(* CODESYS project M241_LexiumILE_minimal_example.project
   Title: M241-ILS2K
   Version: 0.0.0.0
   Author: Philippe

Project tree, tasks and I/O mapping:
  MyController : TM241CE40R, Schneider Electric, order no. TM241CE40R, version 5.1.9.44
    application Application
      libraries: Integrated Lexium Library, 3.2.1.0 (Schneider Electric)
      task MAST (cyclic, interval 20 ms, priority 15, watchdog 100 ms x 1) calls ILE_functionblocks, DISABLE_LIMIT_SWITCH
      global variables GVL
      visualisation Visualization
      program ILE_functionblocks [FBD]
      program DISABLE_LIMIT_SWITCH [SFC]
    DI : Digital Inputs, Schneider Electric, version 5.1.9.44
        input  idwDI_IDW0 : DWORD  // IDW0
        input  ibDI_IB1 : BYTE  // IB1
    DQ : Digital Outputs, Schneider Electric, version 5.1.9.44
        output qwDQ_QW0 : WORD  // QW0
        output qbDQ_QB1 : BYTE  // QB1
    Counters : Counters, Schneider Electric, version 5.1.9.44
    Pulse_Generators : Pulse Generators, Schneider Electric, version 5.1.9.44
    Cartridge_1 : Cartridge, Schneider Electric, version 5.1.9.44
    Cartridge_2 : Cartridge, Schneider Electric, version 5.1.9.44
    IO_Bus : IO bus - TM3, Schneider Electric, version 5.1.9.44
    COM_Bus : COM bus, Schneider Electric, version 5.1.9.44
    Ethernet_1 : Ethernet Network, Schneider Electric, version 5.1.9.44
        settings: IPAddress = [192, 168, 100, 200]; SubnetMask = [255, 255, 255, 0]; GatewayAddress = [192, 168, 100, 254]; WebServer = TRUE; FTP Server = TRUE; SoMachine Protocol = TRUE; Modbus Server = TRUE; NetManage Protocol = TRUE; SNMP protocol = TRUE; Enable Routing = FALSE; WebVisu protocol = TRUE; DHCP Server Active = TRUE; Secured Web Server = TRUE
      Gestionnaire_Ethernet_Industriel : Industrial Ethernet Manager, Schneider Electric, version 1.0.12.40
          settings: BinaryFileSize = 586; Dhcps Host 0.Client Mac Address = [16#00, 16#80, 16#F4, 16#7B, 16#28, 16#E1]; Dhcps Host 0.Client Device Name = 'Lexium-ILx-002'; Dhcps Host 0.Client IP Address = [192, 168, 100, 159]; Dhcps Host 0.Network Mask = [255, 255, 255, 0]; Dhcps Host 0.Default Gateway = [192, 168, 100, 200]; Dhcps Host 2.Client Mac Address = [16#0, 16#0, 16#0, 16#0, 16#0]; Dhcps Host 3.Client Mac Address = [16#0, 16#0, 16#0, 16#0, 16#0]; Dhcps Host 4.Client Mac Address = [16#0, 16#0, 16#0, 16#0, 16#0]; Dhcps Host 5.Client Mac Address = [16#0, 16#0, 16#0, 16#0, 16#0]; Dhcps Host 6.Client Mac Address = [16#0, 16#0, 16#0, 16#0, 16#0]; Dhcps Host 7.Client Mac Address = [16#0, 16#0, 16#0, 16#0, 16#0]; Dhcps Host 8.Client Mac Address = [16#0, 16#0, 16#0, 16#0, 16#0]; Dhcps Host 9.Client Mac Address = [16#0, 16#0, 16#0, 16#0, 16#0]; Dhcps Host 10.Client Mac Address = [16#0, 16#0, 16#0, 16#0, 16#0]; Dhcps Host 11.Client Mac Address = [16#0, 16#0, 16#0, 16#0, 16#0]; Dhcps Host 12.Client Mac Address = [16#0, 16#0, 16#0, 16#0, 16#0]; Dhcps Host 13.Client Mac Address = [16#0, 16#0, 16#0, 16#0, 16#0]; Dhcps Host 14.Client Mac Address = [16#0, 16#0, 16#0, 16#0, 16#0]; Dhcps Host 15.Client Mac Address = [16#0, 16#0, 16#0, 16#0, 16#0]; Dhcps Host 16.Client Mac Address = [16#0, 16#0, 16#0, 16#0, 16#0]; Dhcps Host 17.Client Mac Address = [16#0, 16#0, 16#0, 16#0, 16#0]; Dhcps Host 18.Client Mac Address = [16#0, 16#0, 16#0, 16#0, 16#0]; Dhcps Host 19.Client Mac Address = [16#0, 16#0, 16#0, 16#0, 16#0]; Dhcps Host 20.Client Mac Address = [16#0, 16#0, 16#0, 16#0, 16#0]; Dhcps Host 21.Client Mac Address = [16#0, 16#0, 16#0, 16#0, 16#0]; Dhcps Host 22.Client Mac Address = [16#0, 16#0, 16#0, 16#0, 16#0]; Dhcps Host 23.Client Mac Address = [16#0, 16#0, 16#0, 16#0, 16#0]; Dhcps Host 24.Client Mac Address = [16#0, 16#0, 16#0, 16#0, 16#0]; Dhcps Host 25.Client Mac Address = [16#0, 16#0, 16#0, 16#0, 16#0]; Dhcps Host 26.Client Mac Address = [16#0, 16#0, 16#0, 16#0, 16#0]; Dhcps Host 27.Client Mac Address = [16#0, 16#0, 16#0, 16#0, 16#0]; Dhcps Host 28.Client Mac Address = [16#0, 16#0, 16#0, 16#0, 16#0]; Dhcps Host 29.Client Mac Address = [16#0, 16#0, 16#0, 16#0, 16#0]; Dhcps Host 30.Client Mac Address = [16#0, 16#0, 16#0, 16#0, 16#0]; Dhcps Host 31.Client Mac Address = [16#0, 16#0, 16#0, 16#0, 16#0]; Dhcps Host 32.Client Mac Address = [16#0, 16#0, 16#0, 16#0, 16#0]; Dhcps Host 33.Client Mac Address = [16#0, 16#0, 16#0, 16#0, 16#0]; Dhcps Host 34.Client Mac Address = [16#0, 16#0, 16#0, 16#0, 16#0]; Dhcps Host 35.Client Mac Address = [16#0, 16#0, 16#0, 16#0, 16#0];
            Dhcps Host 36.Client Mac Address = [16#0, 16#0, 16#0, 16#0, 16#0]; Dhcps Host 37.Client Mac Address = [16#0, 16#0, 16#0, 16#0, 16#0]; Dhcps Host 38.Client Mac Address = [16#0, 16#0, 16#0, 16#0, 16#0]; Dhcps Host 39.Client Mac Address = [16#0, 16#0, 16#0, 16#0, 16#0]; Dhcps Host 40.Client Mac Address = [16#0, 16#0, 16#0, 16#0, 16#0]; Dhcps Host 41.Client Mac Address = [16#0, 16#0, 16#0, 16#0, 16#0]; Dhcps Host 42.Client Mac Address = [16#0, 16#0, 16#0, 16#0, 16#0]; Dhcps Host 43.Client Mac Address = [16#0, 16#0, 16#0, 16#0, 16#0]; Dhcps Host 44.Client Mac Address = [16#0, 16#0, 16#0, 16#0, 16#0]; Dhcps Host 45.Client Mac Address = [16#0, 16#0, 16#0, 16#0, 16#0]; Dhcps Host 46.Client Mac Address = [16#0, 16#0, 16#0, 16#0, 16#0]; Dhcps Host 47.Client Mac Address = [16#0, 16#0, 16#0, 16#0, 16#0]; Dhcps Host 48.Client Mac Address = [16#0, 16#0, 16#0, 16#0, 16#0]; Dhcps Host 49.Client Mac Address = [16#0, 16#0, 16#0, 16#0, 16#0]; Dhcps Host 50.Client Mac Address = [16#0, 16#0, 16#0, 16#0, 16#0]; Dhcps Host 51.Client Mac Address = [16#0, 16#0, 16#0, 16#0, 16#0]; Dhcps Host 52.Client Mac Address = [16#0, 16#0, 16#0, 16#0, 16#0]; Dhcps Host 53.Client Mac Address = [16#0, 16#0, 16#0, 16#0, 16#0]; Dhcps Host 54.Client Mac Address = [16#0, 16#0, 16#0, 16#0, 16#0]; Dhcps Host 55.Client Mac Address = [16#0, 16#0, 16#0, 16#0, 16#0]; Dhcps Host 56.Client Mac Address = [16#0, 16#0, 16#0, 16#0, 16#0]; Dhcps Host 57.Client Mac Address = [16#0, 16#0, 16#0, 16#0, 16#0]; Dhcps Host 58.Client Mac Address = [16#0, 16#0, 16#0, 16#0, 16#0]; Dhcps Host 59.Client Mac Address = [16#0, 16#0, 16#0, 16#0, 16#0]; Dhcps Host 60.Client Mac Address = [16#0, 16#0, 16#0, 16#0, 16#0]; Dhcps Host 61.Client Mac Address = [16#0, 16#0, 16#0, 16#0, 16#0]; Dhcps Host 62.Client Mac Address = [16#0, 16#0, 16#0, 16#0, 16#0]; Dhcps Host 63.Client Mac Address = [16#0, 16#0, 16#0, 16#0, 16#0]; Dhcps Host 64.Client Mac Address = [16#0, 16#0, 16#0, 16#0, 16#0]; Dhcps Host 65.Client Mac Address = [16#0, 16#0, 16#0, 16#0, 16#0]; Dhcps Host 66.Client Mac Address = [16#0, 16#0, 16#0, 16#0, 16#0]; Dhcps Host 67.Client Mac Address = [16#0, 16#0, 16#0, 16#0, 16#0]; Dhcps Host 68.Client Mac Address = [16#0, 16#0, 16#0, 16#0, 16#0]; Dhcps Host 69.Client Mac Address = [16#0, 16#0, 16#0, 16#0, 16#0]; Dhcps Host 70.Client Mac Address = [16#0, 16#0, 16#0, 16#0, 16#0]; Dhcps Host 71.Client Mac Address = [16#0, 16#0, 16#0, 16#0, 16#0]; Dhcps Host 72.Client Mac Address = [16#0, 16#0, 16#0, 16#0, 16#0]; Dhcps Host 73.Client Mac Address = [16#0, 16#0, 16#0, 16#0, 16#0]; Dhcps Host 74.Client Mac Address = [16#0, 16#0, 16#0, 16#0, 16#0]; Dhcps Host 75.Client Mac Address = [16#0, 16#0, 16#0, 16#0, 16#0];
            Dhcps Host 76.Client Mac Address = [16#0, 16#0, 16#0, 16#0, 16#0]; Dhcps Host 77.Client Mac Address = [16#0, 16#0, 16#0, 16#0, 16#0]; Dhcps Host 78.Client Mac Address = [16#0, 16#0, 16#0, 16#0, 16#0]; Dhcps Host 79.Client Mac Address = [16#0, 16#0, 16#0, 16#0, 16#0]; Dhcps Host 80.Client Mac Address = [16#0, 16#0, 16#0, 16#0, 16#0]; Dhcps Host 81.Client Mac Address = [16#0, 16#0, 16#0, 16#0, 16#0]; Dhcps Host 82.Client Mac Address = [16#0, 16#0, 16#0, 16#0, 16#0]; Dhcps Host 83.Client Mac Address = [16#0, 16#0, 16#0, 16#0, 16#0]; Dhcps Host 84.Client Mac Address = [16#0, 16#0, 16#0, 16#0, 16#0]; Dhcps Host 85.Client Mac Address = [16#0, 16#0, 16#0, 16#0, 16#0]; Dhcps Host 86.Client Mac Address = [16#0, 16#0, 16#0, 16#0, 16#0]; Dhcps Host 87.Client Mac Address = [16#0, 16#0, 16#0, 16#0, 16#0]; Dhcps Host 88.Client Mac Address = [16#0, 16#0, 16#0, 16#0, 16#0]; Dhcps Host 89.Client Mac Address = [16#0, 16#0, 16#0, 16#0, 16#0]; Dhcps Host 90.Client Mac Address = [16#0, 16#0, 16#0, 16#0, 16#0]; Dhcps Host 91.Client Mac Address = [16#0, 16#0, 16#0, 16#0, 16#0]; Dhcps Host 92.Client Mac Address = [16#0, 16#0, 16#0, 16#0, 16#0]; Dhcps Host 93.Client Mac Address = [16#0, 16#0, 16#0, 16#0, 16#0]; Dhcps Host 94.Client Mac Address = [16#0, 16#0, 16#0, 16#0, 16#0]; Dhcps Host 95.Client Mac Address = [16#0, 16#0, 16#0, 16#0, 16#0]; Dhcps Host 96.Client Mac Address = [16#0, 16#0, 16#0, 16#0, 16#0]; Dhcps Host 97.Client Mac Address = [16#0, 16#0, 16#0, 16#0, 16#0]; Dhcps Host 98.Client Mac Address = [16#0, 16#0, 16#0, 16#0, 16#0]; Dhcps Host 99.Client Mac Address = [16#0, 16#0, 16#0, 16#0, 16#0]; Dhcps Host 100.Client Mac Address = [16#0, 16#0, 16#0, 16#0, 16#0]; Dhcps Host 101.Client Mac Address = [16#0, 16#0, 16#0, 16#0, 16#0]; Dhcps Host 102.Client Mac Address = [16#0, 16#0, 16#0, 16#0, 16#0]; Dhcps Host 103.Client Mac Address = [16#0, 16#0, 16#0, 16#0, 16#0]; Dhcps Host 104.Client Mac Address = [16#0, 16#0, 16#0, 16#0, 16#0]; Dhcps Host 105.Client Mac Address = [16#0, 16#0, 16#0, 16#0, 16#0]; Dhcps Host 106.Client Mac Address = [16#0, 16#0, 16#0, 16#0, 16#0]; Dhcps Host 107.Client Mac Address = [16#0, 16#0, 16#0, 16#0, 16#0]; Dhcps Host 108.Client Mac Address = [16#0, 16#0, 16#0, 16#0, 16#0]; Dhcps Host 109.Client Mac Address = [16#0, 16#0, 16#0, 16#0, 16#0]; Dhcps Host 110.Client Mac Address = [16#0, 16#0, 16#0, 16#0, 16#0]; Dhcps Host 111.Client Mac Address = [16#0, 16#0, 16#0, 16#0, 16#0]; Dhcps Host 112.Client Mac Address = [16#0, 16#0, 16#0, 16#0, 16#0]; Dhcps Host 113.Client Mac Address = [16#0, 16#0, 16#0, 16#0, 16#0]; Dhcps Host 114.Client Mac Address = [16#0, 16#0, 16#0, 16#0, 16#0]; Dhcps Host 115.Client Mac Address = [16#0, 16#0, 16#0, 16#0, 16#0];
            Dhcps Host 116.Client Mac Address = [16#0, 16#0, 16#0, 16#0, 16#0]; Dhcps Host 117.Client Mac Address = [16#0, 16#0, 16#0, 16#0, 16#0]; Dhcps Host 118.Client Mac Address = [16#0, 16#0, 16#0, 16#0, 16#0]; Dhcps Host 119.Client Mac Address = [16#0, 16#0, 16#0, 16#0, 16#0]; Dhcps Host 120.Client Mac Address = [16#0, 16#0, 16#0, 16#0, 16#0]; Dhcps Host 121.Client Mac Address = [16#0, 16#0, 16#0, 16#0, 16#0]; Dhcps Host 122.Client Mac Address = [16#0, 16#0, 16#0, 16#0, 16#0]; Dhcps Host 123.Client Mac Address = [16#0, 16#0, 16#0, 16#0, 16#0]; Dhcps Host 124.Client Mac Address = [16#0, 16#0, 16#0, 16#0, 16#0]; Dhcps Host 125.Client Mac Address = [16#0, 16#0, 16#0, 16#0, 16#0]; Dhcps Host 126.Client Mac Address = [16#0, 16#0, 16#0, 16#0, 16#0]; Dhcps Host 127.Client Mac Address = [16#0, 16#0, 16#0, 16#0, 16#0]; Dhcps Host 128.Client Mac Address = [16#0, 16#0, 16#0, 16#0, 16#0]; serialized Values = 010bc991-f7f9-45b2-8b15-1d199ae18604=0|; InterfaceUsedByDhcpSize = 4; InterfaceUsedByDhcp = [192,168,100,200]
          unmapped channels: Global Status, Healthbit 0, Healthbit 1, Healthbit 2, Healthbit 3, Channels 0, Channels 1, Channels 2, Channels 3
        Lexium_ILE : Lexium ILE, Schneider Electric, order no. 89330, version 1.2.11.0
            settings: IP address of Target = [192,168,100,159]; MAC address of Target = [16#00, 16#80, 16#F4, 16#7B, 16#28, 16#E1]; DeviceNumber = 1; Object Input1 = [0, 40, 268500992, 257]; Object Output1 = [1, 40, 268566528, 257]; Connection Id List = [257,0,0,0,0,0,0,0]; Connection Settings.Connection Number = 257
            unmapped channels: Input Read/Write IclA, Output Read/Write IclA
    Serial_Line_1 : Serial line, Schneider Electric, version 5.1.9.44
      SoMachine_Network_Manager : Machine Expert-Network Manager, Schneider Electric, version 4.0.0.4
    Serial_Line_2 : Serial line, Schneider Electric, version 5.1.9.44
      Modbus_Manager : Modbus Manager, Schneider Electric, version 4.0.0.4
  libraries: VisuSymbols, 3.5.10.0 (System)
  text list GlobalTextList
*)

// MyController/Application/GVL

VAR_GLOBAL
	ILE_Disable_switch_neg,ILE_Disable_switch_neg_OK:BOOL;
	ILE_Disable_switch_pos,ILE_Disable_switch_pos_OK:BOOL;
	
	
	ILE_Power, ILE_Power_OK: BOOL;
	ILE_Reset, ILE_Reset_OK: BOOL;
	
	MC_status_read:BOOL;
	DisableOK:BOOL;
	
	
	Power1: GIPLC.MC_Power;
	MC_Reset_0: GIPLC.MC_Reset;
	reset0: BOOL;
	valeur3: WORD;
	MC_MoveRelative_0: GIPLC.MC_MoveRelative;
	movement0: BOOL;
	distance: DINT;
	vitesse: DINT;
	dist: INT;
	erreur0: BOOL;
	err_type: BOOL;
	err_id: WORD;
	err_axisid: WORD;
	MC_ReadAXiserror: GIPLC.MC_ReadAxisError;
	MC_WriteParameter_ILX_0: GIPLC.MC_WriteParameter;
	MC_WriteParameter_0: GIPLC.MC_WriteParameter;
	SetLimitSwitch_ILX_0: GILXM.SetLimitSwitch_ILX;
	SetLimitSwitch_ILX: GILXM.SetLimitSwitch_ILX;
	SetLimitSwitch_ILX_pos: GILXM.SetLimitSwitch_ILX;
	SetLimitSwitch_ILX_neg: GILXM.SetLimitSwitch_ILX;
	MC_ReadActualPosition: GIPLC.MC_ReadActualPosition;
	mesure: BOOL;
	
END_VAR

// MyController/Application/ILE_functionblocks
PROGRAM ILE_functionblocks
VAR
	MC_ReadStatus_0: GIPLC.MC_ReadStatus;
END_VAR

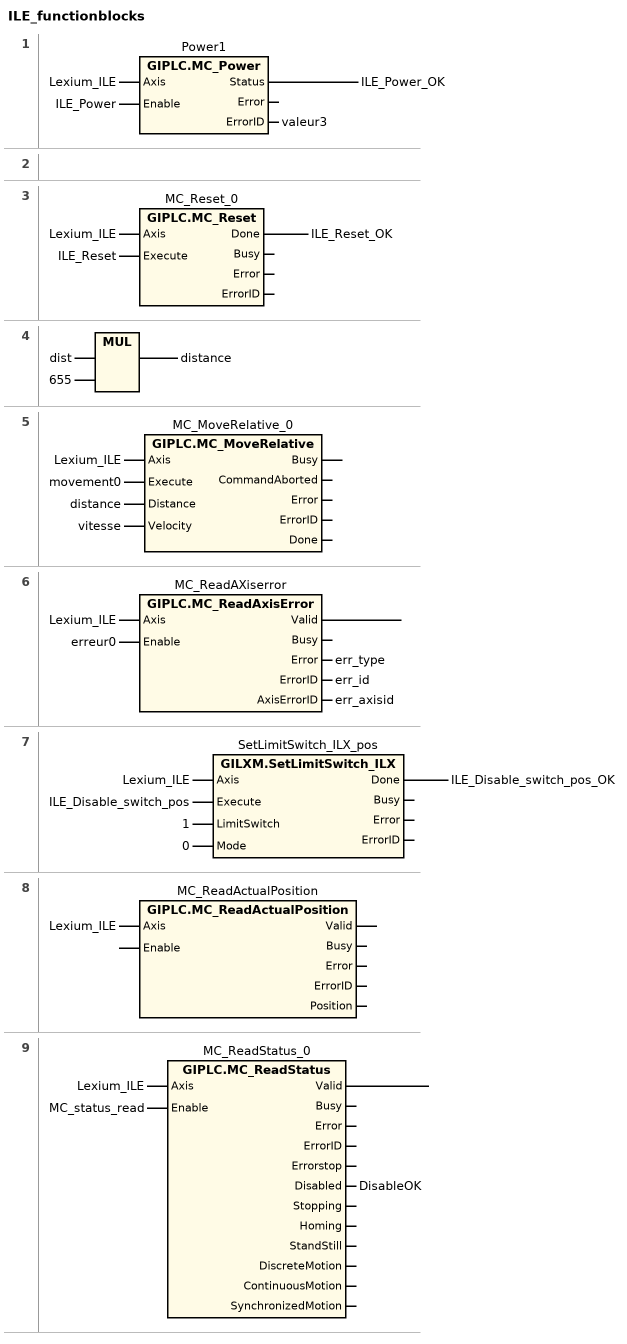
// NETWORK 1
Power1(Axis := Lexium_ILE, Enable := ILE_Power, ErrorID => valeur3); // GIPLC.MC_Power
ILE_Power_OK := Power1.Status;

// NETWORK 2

// NETWORK 3
MC_Reset_0(Axis := Lexium_ILE, Execute := ILE_Reset); // GIPLC.MC_Reset
ILE_Reset_OK := MC_Reset_0.Done;

// NETWORK 4
distance := dist * 655;

// NETWORK 5
MC_MoveRelative_0(Axis := Lexium_ILE, Execute := movement0, Distance := distance, Velocity := vitesse); // GIPLC.MC_MoveRelative

// NETWORK 6
MC_ReadAXiserror(
    Axis := Lexium_ILE,
    Enable := erreur0,
    Error => err_type,
    ErrorID => err_id,
    AxisErrorID => err_axisid); // GIPLC.MC_ReadAxisError

// NETWORK 7
SetLimitSwitch_ILX_pos(Axis := Lexium_ILE, Execute := ILE_Disable_switch_pos, LimitSwitch := 1, Mode := 0); // GILXM.SetLimitSwitch_ILX
ILE_Disable_switch_pos_OK := SetLimitSwitch_ILX_pos.Done;

// NETWORK 8
MC_ReadActualPosition(Axis := Lexium_ILE); // GIPLC.MC_ReadActualPosition

// NETWORK 9
MC_ReadStatus_0(Axis := Lexium_ILE, Enable := MC_status_read, Disabled => DisableOK); // GIPLC.MC_ReadStatus

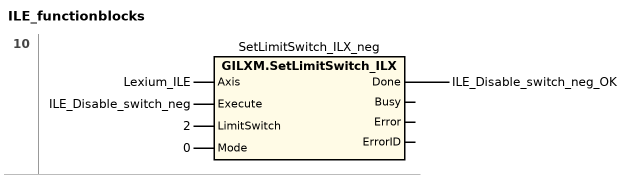
// NETWORK 10
SetLimitSwitch_ILX_neg(Axis := Lexium_ILE, Execute := ILE_Disable_switch_neg, LimitSwitch := 2, Mode := 0); // GILXM.SetLimitSwitch_ILX
ILE_Disable_switch_neg_OK := SetLimitSwitch_ILX_neg.Done;

END_PROGRAM

// MyController/Application/DISABLE_LIMIT_SWITCH
PROGRAM DISABLE_LIMIT_SWITCH
VAR
END_VAR

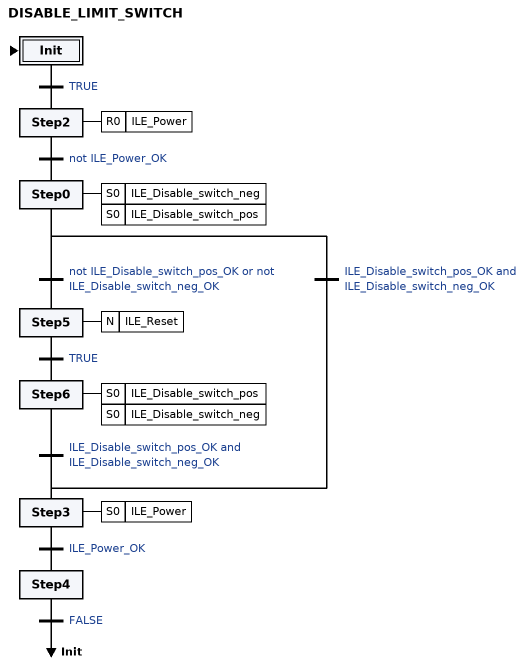
INITIAL_STEP Init:
END_STEP
TRANSITION FROM Init TO Step2
    := TRUE;
END_TRANSITION
STEP Step2:
    ILE_Power(R0);
END_STEP
TRANSITION FROM Step2 TO Step0
    := not ILE_Power_OK;
END_TRANSITION
STEP Step0:
    ILE_Disable_switch_neg(S0);
    ILE_Disable_switch_pos(S0);
END_STEP
TRANSITION FROM Step0 TO Step5
    := not ILE_Disable_switch_pos_OK or not ILE_Disable_switch_neg_OK;
END_TRANSITION
STEP Step5:
    ILE_Reset(N);
END_STEP
TRANSITION FROM Step5 TO Step6
    := TRUE;
END_TRANSITION
STEP Step6:
    ILE_Disable_switch_pos(S0);
    ILE_Disable_switch_neg(S0);
END_STEP
TRANSITION FROM Step6 TO Step3
    := ILE_Disable_switch_pos_OK and ILE_Disable_switch_neg_OK;
END_TRANSITION
TRANSITION FROM Step0 TO Step3
    := ILE_Disable_switch_pos_OK and ILE_Disable_switch_neg_OK;
END_TRANSITION
STEP Step3:
    ILE_Power(S0);
END_STEP
TRANSITION FROM Step3 TO Step4
    := ILE_Power_OK;
END_TRANSITION
STEP Step4:
END_STEP
TRANSITION FROM Step4 TO Init
    := FALSE;
END_TRANSITION

END_PROGRAM

// MyController/Application/Visualization
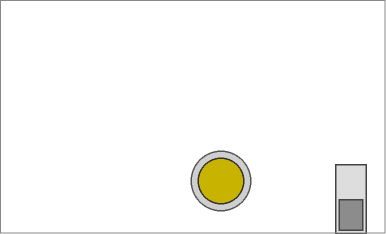
VISUALIZATION Visualization  // 386x234
    Lamp1 (186,146 70x70), variable: ILE_functionblocks.power, style: Lamp-Lamp1-Yellow
    DipSwitch (316,164 70x70), behaviour: TOGGLE, style: Switch-DipSwitch-Gray
END_VISUALIZATION
